(* PLC project Unnamed, Unknown Unnamed 1 *)
(* stored: creationDateTime 2026-08-28T18:13:26, modificationDateTime 2026-08-28T18:13:26 *)

PROGRAM main
  VAR
    myVar : REAL;
    counter : INT;
    total : REAL;
    gate : BOOL;
    mode : INT;
    result : REAL;
    i : INT;
  END_VAR

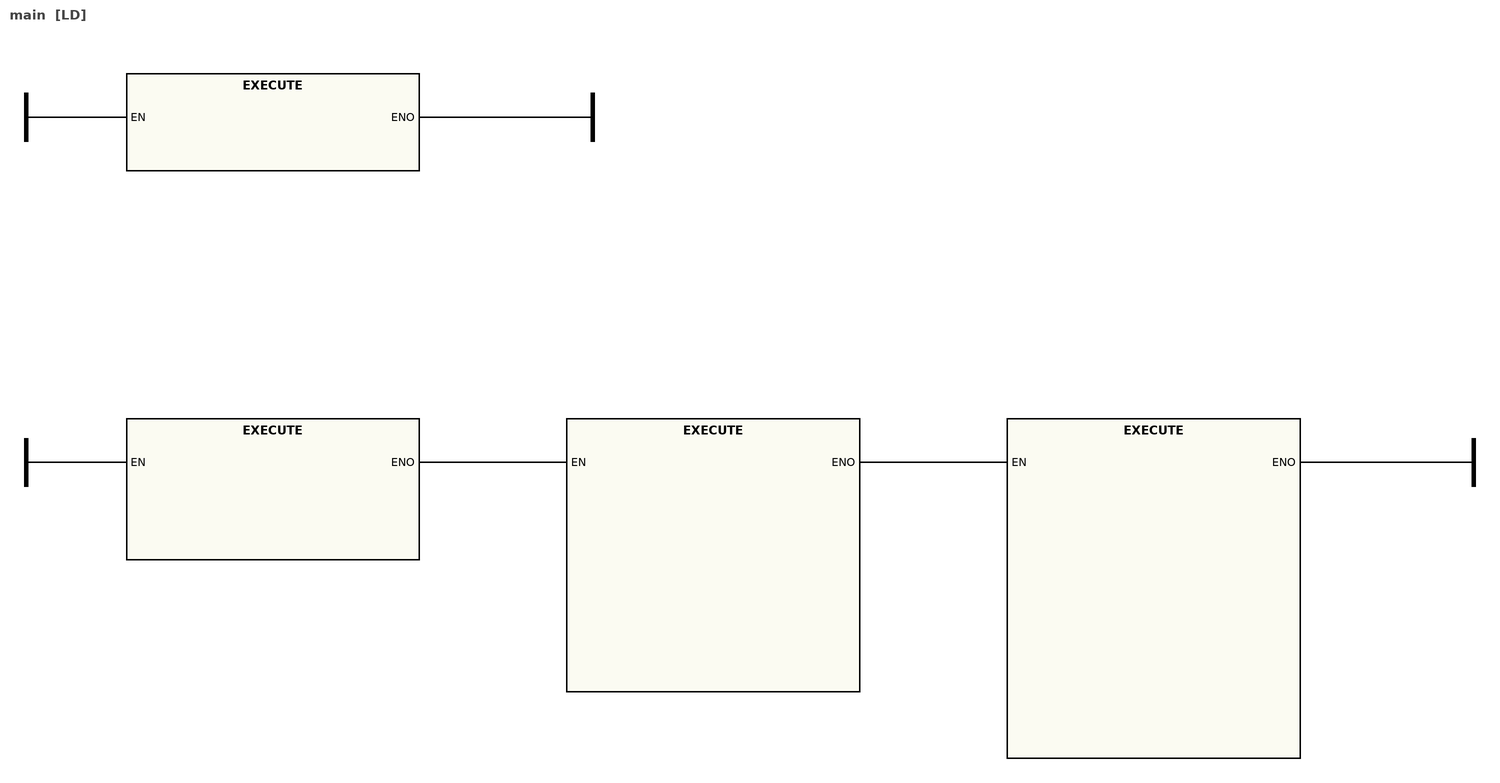
(* LD diagram, written out as Structured Text *)
myVar := myVar + 0.01;
counter := counter + 1;
total := total + 0.01;
result := total * 2.0;
IF counter > 100 THEN
    counter := 0;
ELSIF counter < 0 THEN
    counter := 100;
END_IF;

IF total <> 0.0 AND gate THEN
    result := total / 2.0;
END_IF;
total := 0.0;
FOR i := 1 TO 10 BY 1 DO
    total := total + REAL#1.5;
END_FOR;

CASE mode OF
    0: result := 0.0;
    1, 2: result := total;
    3..5: result := total * 2.0;
ELSE
    result := -1.0;
END_CASE;
END_PROGRAM

PROGRAM test_FBD
  VAR
    myVar : REAL;
    myOut : BOOL;
  END_VAR

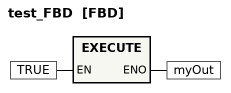
(* FBD diagram, written out as Structured Text *)
IF TRUE THEN
  myVar := myVar + 0.01;
END_IF;
myOut := TRUE;
END_PROGRAM

CONFIGURATION Config0
  RESOURCE Res0 ON PLC
    TASK task0(INTERVAL := T#20ms, PRIORITY := 1);
    PROGRAM instance0 WITH task0 : main;
    PROGRAM instance1 WITH task0 : test_FBD;
  END_RESOURCE
END_CONFIGURATION
